FUNCTION_BLOCK FB_WorkerDefGrid_Print_WEU EXTENDS FB_WorkerDefGrid IMPLEMENTS I_PrintSubsystem
VAR_INPUT
  nPrintPos             : DINT;   // Absolute printing position [SubPx]
  fMasterSpeed          : LREAL;  // Speed [m/s]
  bHardwareSync         : BOOL;   // hw sync signal (chenerates a triger internally)
  bHardwareHold         : BOOL;   // hw hold signal
  fPrintStartOffset     : LREAL;  // X-Shift StartOffset from Module reference (configurative PU/PM/PG/PA ADS offset) [m]
  fPrintYOffset         : LREAL;  // Y-Shift
  // fine alignement live parameter
  fPUElevation          : LREAL;  // PU distance from substrate [m]
END_VAR
VAR
  // print
  // - references
  _pAdsPg            : POINTER TO ST_ADS_PG;      // pg ads reference (for pa)
  // - instances
  fbPs               : FB_PS_Grid;
  fbPa               : FB_PA;
  fB_PcAdapter       : FB_PC_Adapter;
  
  // grid specific
  // - references
  _iParamMediator    : I_ParamMediator;
  // - settings
  sDefGridSettings   : ST_DefGridSettings; 
  // - state 
  fCurrentColumnPos  : LREAL; // Currently column position
  fCurrentPreCharge  : LREAL; // Currently to be precharged
  nChargedColumns    : UDINT; // Already charged columns


  // print corrections
  nPointCorrections  : UDINT;     // number of registered point correction handler
  iPointCorrections  : ARRAY[1..nC_NUM_POINTCORRECTIONS] OF I_GridPointCorrection;  // point corrections
  
  // - Time of flight correction of droplets
  fbDropSpeedComp    : FB_DropSpeedComp;
  //
  _pAdsCam           : POINTER TO ST_ADS_CAMERA;  // camera interface PUC
  // - global shifts (applied globally and not on every single point (calcualted based on all CT points))
  _fDxGlobalShift    : LREAL;
  _fDyGlobalShift    : LREAL;

  // settings or helper
  _fPrintStartOffset : LREAL;   // internal print start offset (distance Cam -> PG1 + PG Offset + PU offset)
  _nPosX0            : DINT;    // X0 for last attached CT (detected postion)
  _nPosXS            : DINT;    // XS for last attached CT (shifted print start position)
  _nPosXDelta        : DINT;    // Shift value X0 -> XS
  _fPosY             : LREAL;   // Y shift for last attached CT
  _nPosDeltaToPrint  : DINT;    // delta pos in [SbuPx] from attach to print
  _sCurrentImgDepth  : LREAL;   // Job: current image length [m]
  _bEndless          : BOOL;    // Job: endless
  _bPaStarted        : BOOL;
  _bPaStartRequested : BOOL;
  _sJobDef           : BOOL;
  fBStartTimeout     : TON;
  rTrigHwSync        : R_TRIG;
  _bForceDefGridOff  : BOOL;    // force deformation grid stream to ph off (send 0)
  
  (*grid limit*)
  _fLimitCorrectionX : LREAL;     // correction limit in y (abs) [px]
  _fLimitCorrectionY : LREAL;     // correction limit in y (abs) [px]
    
  (*Messaging*)
  (*we could implement a message handler for ST_ADS_PG message interface*)

END_VAR

VAR PERSISTENT
  _fColumnsToPrecharge : LREAL := nC_COLUMNS_TO_PRECHARGE;
  _fStartShiftOffset   : LREAL := fC_START_SHIFT_OFFSET;
  _fStartShiftFactor   : LREAL := fC_START_SHIFT_FACTOR;
END_VAR

VAR CONSTANT
  iC_NUM_MSG               : UDINT := 5;
  nC_COLUMNS_TO_PRECHARGE  : LREAL := 2.1;
  fC_GRIDPOINT_STREAM_TIME : LREAL := 0.0025;     // time to stream one point [s]
  fC_START_SHIFT_FACTOR    : LREAL := -2.4E-2;
  fC_START_SHIFT_OFFSET    : LREAL := -1.0E-2;
  nC_NUM_POINTCORRECTIONS  : UDINT := 5;
END_VAR

(*
DOC:
What will be different to FB_WorkerDefGrid_Print of DMAX
- Re-Sync StartPosDetect interface with optional camera data (y-shift)
  Clear with Attach(), security clearance
- (maybe not needed) Stream grid faster to PC (we have no break for switching the CT in endless)
- New PDI StartPostion update (+print start only for first CT) --> send to NIOS or hw buffer
- PDI GridPoint stream
- New PDI PrintingLength update (after last streamed point)
- Other rules for Worker position calculation
*)

PROPERTY aPaState : STRING
GET
aPaState := fbPa.aPaState;
END_GET
END_PROPERTY

METHOD PROTECTED  Attach : BOOL
VAR_INPUT
  iCT              : I_CT;                         (*container at triggered event position*)
END_VAR
Attach:=FALSE;

IF SUPER^.Attach(iCT:=iCT) THEN
  // Additional worker checks
    // - job is valid?
  IF _pAttachedCt^.pJob = 0 OR NOT _bJobActive THEN
    Release(iCT:=iCT);
    RETURN;   // do not print
  
  // CT valid & CT present
  ELSIF NOT _pAttachedCt^.bValid OR NOT _pAttachedCt^.bProductPresent THEN
    Release(iCT:=iCT);
    RETURN;   // do not print
  
  // Ignore start due to hardware hold  
  ELSIF bHardwareHold THEN
    _pAttachedCt^.setError(ErrDef:=EC_Print.ecPaAbortHold, Src:=_pEcSrc^);
    Release(iCT:=iCT);
    RETURN;   // do not print
  
  // - OK attach
  ELSE
    Attach := TRUE;
	END_IF
  
  
  //Prepare print station
  sDefGridSettings := _iParamMediator.sDeformationGridSetttings; // or get from CT (but needs to be set even if WorkerDeformation is not enabled) _pAttachedCt^.sDefGridSettings;
  // fix some potential errors
  IF sDefGridSettings.nGridPitchX = 0 THEN sDefGridSettings.nGridPitchX :=1024; LogError(F_concat2('grid not configured, set default nGridPitchX=',TO_STRING(sDefGridSettings.nGridPitchX))); END_IF
  IF sDefGridSettings.nGridPitchY = 0 THEN sDefGridSettings.nGridPitchY :=1024; LogError(F_concat2('grid not configured, set default nGridPitchY=',TO_STRING(sDefGridSettings.nGridPitchY))); END_IF
  
  nChargedColumns := 0;
  fbPs.bPrintEnable := iCT.bValid AND iCT.bProductPresent;
  fbPs.setGrid(sGrid:=sDefGridSettings);
  _fDxGlobalShift := _pAttachedCt^.fDxShift;
  _fDyGlobalShift := _pAttachedCt^.fDyShift;

  //Start print, PA should be in READY or DONE
  
  // Set X print position
  _nPosX0 :=    _pAttachedCt^.getPosX0(nPosDomain:=E_PosDomain.master_pos)
              //- General Shift
              - F_MeterToSubPixel(fbDropSpeedComp.fDropPlacementError, _fPrintResolution*_fSubPxResolution); // - drop compensation*)
  _nPosXDelta := F_MeterToSubPixel(_fPrintStartOffset, _fPrintResolution*_fSubPxResolution); // + PG/PA Shift (additional PG offset 0 for firstLine)
  
  IF GVL_Deformation.bC_UseGlobalGridShift THEN
    _nPosXDelta := _nPosXDelta + FC_LREAL_TO_DINT(_fDxGlobalShift);                  // + global shift from grid points
  END_IF

  _nPosXS := _nPosX0 + _nPosXDelta;
  fB_PcAdapter.setPrintStartPos(nX0:=_nPosXS);
  
  // Set Y print position
  _fPosY := fPrintYOffset;
  IF GVL_Deformation.bC_UseGlobalGridShift THEN
    _fPosY := _fPosY + _fDyGlobalShift;    // + global shift from grid points
  END_IF
  fB_PcAdapter.setPrintYShift(nYShift:=FC_LREAL_TO_DINT(_fPosY));

  // check
  IF _nPosXS < nPrintPos THEN
    LogWarning(Msg:=F_Concat4('Print start position:', TO_STRING(_nPosXS) ,' < Encoder position:', TO_STRING(nPrintPos)));
	END_IF
  
  // save current distance to print position
  _nPosDeltaToPrint := _nPosXS - iCT.GetPos(nPosDomain:=E_PosDomain.master_pos) - _nPosX0;
  checkGridTiming();
  
  
  IF NOT fbPa.bPrinting THEN   // fB_PcAdapter.bAllPrinting
    IF NOT fbPa.printStart() THEN
      LogError(Msg:='PA not ready to start at attach');
      Release(iCT := iCT);
    ELSE
      _bPaStarted := FALSE;
      _bPaStartRequested := TRUE;
      Attach:=TRUE;
    END_IF
  ELSE
    // update start postion if it was already started (endless)
    {warning 'TODO: implement print restart in endless'}
    //fbPa.restartPrint();
    Attach:=TRUE;
  END_IF
  
  // debug log
  LogLvl(Lvl:=E_LogSeverity.Debug, F_Concat4('printStart: at XS:', TO_STRING(_nPosXS), ' ', _pAttachedCt^.print(0)));  // print container
  IF GVL_Deformation.bC_UseGlobalGridShift THEN
    LogLvl(Lvl:=E_LogSeverity.Debug, F_Concat4(
                                        F_Concat3('> XS = X0(', TO_STRING(_pAttachedCt^.GetPosX0(nPosDomain:=E_PosDomain.master_pos)), ')'),
                                        F_Concat3(' + shDx(', TO_STRING(_fDxGlobalShift), ')'),
                                        F_Concat3(' + shStartOffs(', TO_STRING(F_MeterToSubPixel(_fPrintStartOffset,_fPrintResolution*_fSubPxResolution)), ')'),
                                        F_Concat3(' - shDropComp(', TO_STRING(F_MeterToSubPixel(fbDropSpeedComp.fDropPlacementError,_fPrintResolution*_fSubPxResolution)), ')')
                                     ));
  ELSE
    LogLvl(Lvl:=E_LogSeverity.Debug, F_Concat3(
                                        F_Concat3('> XS = X0(', TO_STRING(_pAttachedCt^.GetPosX0(nPosDomain:=E_PosDomain.master_pos)), ')'),
                                        F_Concat3(' + shStartOffs:', TO_STRING(F_MeterToSubPixel(_fPrintStartOffset,_fPrintResolution*_fSubPxResolution)), ')'),
                                        F_Concat3( ' - shDropComp:', TO_STRING(F_MeterToSubPixel(fbDropSpeedComp.fDropPlacementError,_fPrintResolution*_fSubPxResolution)), ')')
                                     ));
  END_IF
  
  
ELSE
  // parent attach failed case
END_IF
END_METHOD

PROPERTY bPausePrintCanEx : BOOL
GET
bPausePrintCanEx := FALSE; //Not implemented
END_GET
END_PROPERTY

PROPERTY bPcEnabled : BOOL
GET
bPcEnabled := fB_PcAdapter.bPcEnable;
END_GET
END_PROPERTY

PROPERTY bPrintEnabled : BOOL
GET
bPrintEnabled := _bEnable;
END_GET
END_PROPERTY

PROPERTY bPrintError : BOOL
GET
bPrintError := bError; // Worker error 
                  // or fB_PcAdapter.bError
END_GET
END_PROPERTY

PROPERTY bPrinting : BOOL
GET
bPrinting := fbPa.bPrinting;
END_GET
END_PROPERTY

PROPERTY bPrintReady : BOOL
GET
bPrintReady := fbPa.bReady;
END_GET
END_PROPERTY

PROPERTY bStartPrintCanEx : BOOL
GET
bStartPrintCanEx := fbPa.bStartCanEx;
END_GET
END_PROPERTY

PROPERTY bStopPrintCanEx : BOOL
GET
bStopPrintCanEx := fbPa.bStopCanEx;
END_GET
END_PROPERTY

{attribute 'monitoring':='call'}
PROPERTY bWorkerEnable : BOOL
GET
bWorkerEnable := SUPER^.bWorkerEnable;
END_GET
SET
IF _pAdsPg = 0 THEN
  SUPER^.bWorkerEnable := bWorkerEnable;
ELSE
  // mask worker enable with group enable
  SUPER^.bWorkerEnable := bWorkerEnable AND _pAdsPg^.bI_Enable;  
END_IF
END_SET
END_PROPERTY

METHOD PRIVATE checkGridTiming : BOOL
VAR
END_VAR
// check for timing problems
IF fMasterSpeed <> 0 THEN

  // - check pre-charge at beginning
  IF _fColumnsToPrecharge * fC_GRIDPOINT_STREAM_TIME * GVL_Deformation.nC_GridRoiRows >= F_SubPixelToMeter(lPosSubPx:=_nPosDeltaToPrint, fResSubPx:=_fPrintResolution*_fSubPxResolution) / fMasterSpeed  THEN
       LogError('Machine too fast for grid stream (for pre-charge at attach)');
  END_IF
  
 // - check charge time needed per columns vs machine speed and grid-sizeY
 IF GVL_Deformation.nC_GridRoiRows * fC_GRIDPOINT_STREAM_TIME >= F_SubPixelToMeter(lPosSubPx:=TO_DINT(sDefGridSettings.nGridPitchX), fResSubPx:=_fPrintResolution) / fMasterSpeed THEN
   LogError('Machine too fast for grid stream (time rows per column)');
 END_IF

END_IF
END_METHOD

(*
  Limit correction to boundaries
  :return: TRUE if limited
*)
METHOD PRIVATE correctionLimit : BOOL
VAR_INPUT
  pPoint : POINTER TO ST_DeformationPointAccurate;
END_VAR
VAR
  bLimited : BOOL;
  nExeedX, nExeedY : LREAL;
END_VAR
// limit point correction to boundaries and inform
IF    pPoint^.dx >= _fLimitCorrectionX    THEN nExeedX := pPoint^.dx; pPoint^.dx := _fLimitCorrectionX;    bLimited:=TRUE; 
ELSIF pPoint^.dx <= -1*_fLimitCorrectionX THEN nExeedX := pPoint^.dx; pPoint^.dx := -1*_fLimitCorrectionX; bLimited:=TRUE;
ELSIF pPoint^.dy >= _fLimitCorrectionY    THEN nExeedY := pPoint^.dy; pPoint^.dy := _fLimitCorrectionY;    bLimited:=TRUE;
ELSIF pPoint^.dy <= -1*_fLimitCorrectionY THEN nExeedY := pPoint^.dy; pPoint^.dy := -1*_fLimitCorrectionY; bLimited:=TRUE;
END_IF
IF bLimited THEN 
  LogLvl(Lvl:=E_LogSeverity.Warning, Msg:=F_Concat5( 'Point=',TO_STRING(pPoint^.index),
                                                     F_Concat5(' c/r(',TO_STRING(pPoint^.col),'/',TO_STRING(pPoint^.row), ') '),
                                                     F_Concat4('dx:', TO_STRING(nExeedX), ' dy:', TO_STRING(nExeedY)),
                                                     ' correction exceeded limit')); 
END_IF
correctionLimit := bLimited;
END_METHOD

METHOD PRIVATE correctionUpdate : BOOL
VAR_INPUT
  pPoint : POINTER TO ST_DeformationPointAccurate;
END_VAR
VAR
  i : UDINT;
END_VAR

// here apply all PU specific corrections
// - mechanical stretch based on temperature extension (if not done in Camera)
// - banana correction
// - Y-shifts of PU
// - trapzedoial correction
// - ...

// global dx/dy correction
//   remove global shift from GridPoints (shifted by PU)
IF GVL_Deformation.bC_UseGlobalGridShift THEN
  pPoint^.dx := pPoint^.dx - _fDxGlobalShift;
  pPoint^.dy := pPoint^.dy - _fDyGlobalShift;
END_IF

// PU Deformation correction
IF GVL_Deformation.bC_UsePUDeformation THEN
  FOR i:=1 TO nPointCorrections DO
    iPointCorrections[i].updateCorrection(pPoint:=pPoint);
  END_FOR
END_IF
END_METHOD

(*
  Max. supported speed [m/s], 0 if not available
*)
{attribute 'monitoring':='call'}
PROPERTY fMaxSpeed : LREAL
GET
VAR
  nSpeedMpMin : DINT;
END_VAR
nSpeedMpMin := SEL(bWorkerEnable AND _pAdsPg <> 0, 0, _pAdsPg^.sI_MaxPrintSpeed.lI_Val);
fMaxSpeed := TO_LREAL(nSpeedMpMin)/60;
END_GET
END_PROPERTY

{attribute 'monitoring':='call'}
PROPERTY fStartShiftFactor : LREAL
GET
fStartShiftFactor := _fStartShiftFactor;
END_GET
SET
_fStartShiftFactor := fStartShiftFactor;
END_SET
END_PROPERTY

{attribute 'monitoring':='call'}
PROPERTY fStartShiftOffset : LREAL
GET
fStartShiftOffset := _fStartShiftOffset;
END_GET
SET
_fStartShiftOffset := fStartShiftOffset;
END_SET
END_PROPERTY

METHOD PROTECTED gridUpdate : BOOL
VAR_INPUT
  bEnableDeformation : BOOL;      // enable correction update, else correction (0/0) is written
END_VAR
VAR
  sPoint : ST_DeformationPointAccurate;
  nRow : UDINT;
  nAvailPoints : UDINT;
  nConvErr : UDINT;
END_VAR
VAR_INST
  nAvailPoints_mem : UDINT;
END_VAR
//TODO: rewrite this method to look cleaner (less if else)
IF sDefGridSettings.nGridSizeX = 0 THEN RETURN; END_IF          // avoid endless loops
IF sDefGridSettings.nGridSizeY = 0 THEN RETURN; END_IF

gridUpdate:=TRUE;

// calculate grid column position
IF sDefGridSettings.nGridPitchX <> 0 THEN
  fCurrentColumnPos := fCtPosition / (sDefGridSettings.nGridPitchX * _fSubPxResolution);   // calc grid column position relative to worker
END_IF

//Check for next correction update 
IF fCurrentColumnPos + _fColumnsToPrecharge > nChargedColumns AND nChargedColumns <= sDefGridSettings.nGridSizeX THEN
  fCurrentPreCharge := fCurrentColumnPos + _fColumnsToPrecharge;
  IF bEnableDeformation THEN 
    // sync deformation points
    WHILE FLOOR(fCurrentPreCharge) > nChargedColumns AND nChargedColumns <= sDefGridSettings.nGridSizeX DO
      nAvailPoints := _pAttachedCt^.nAvailableGridPoints;
      IF nAvailPoints >= sDefGridSettings.nGridSizeY * (nChargedColumns+1) THEN // Complete column available?
        nAvailPoints_mem := 0;
        LogLvl(Lvl:=E_LogSeverity.Debug, Msg:=F_Concat2('Charge CG col: ',TO_STRING(nChargedColumns)));
        FOR nRow := 0 TO sDefGridSettings.nGridSizeY - 1 DO
          // get points
          IF _pAttachedCt^.getDeformationPoint(nCol:=nChargedColumns, nRow:=nRow, sPoint => sPoint) THEN
            // transfer the displacement into a correction
            sPoint.dx := sPoint.dx;   // nothing to change
            sPoint.dy := sPoint.dy;
            
            // apply PU corrections
            correctionUpdate(pPoint:=ADR(sPoint));
            
            // correction limitation
            correctionLimit(pPoint:=ADR(sPoint));
            
            // send point
            IF NOT fbPs.newGridPoint(sPoint:=sPoint) THEN
               LogError(Msg:='stream new point failed');
               gridUpdate:=FALSE;
               RETURN;
            END_IF
          ELSE
            LogError(Msg:='get new grid point failed');
            gridUpdate:=FALSE;
          END_IF
        END_FOR
        
        nChargedColumns := nChargedColumns + 1;
      ELSE
        IF nAvailPoints > nAvailPoints_mem THEN // log once or after every update of new available poinst
          LogError(Msg:='point column expected but not available');
        END_IF
        nAvailPoints_mem := nAvailPoints;
        gridUpdate:=FALSE;
        RETURN;
      END_IF 
    END_WHILE
  ELSE
    // send points with no deformation
    FOR nRow := 0 TO sDefGridSettings.nGridSizeY - 1 DO
        MEMSET(destAddr:=ADR(sPoint), fillByte:=0, n:=SIZEOF(sPoint));
        sPoint.col := TO_DINT(nChargedColumns);
        sPoint.row := TO_DINT(nRow);
        IF NOT fbPs.newGridPoint(sPoint:=sPoint) THEN
           LogError(Msg:='stream new point failed');
           gridUpdate:=FALSE;
           RETURN;
        END_IF
    END_FOR
    nChargedColumns := nChargedColumns + 1;
  END_IF
END_IF
END_METHOD

METHOD InitWorkerPrint : BOOL
VAR_INPUT
  pAdsPg                : POINTER TO ST_ADS_PG;       // pg ads reference (worker prints ads)
  iDefGridParamMediator : I_ParamMediator;            // for deformation settings
  fLimitCorrectionX     : LREAL;                      // correction limit in y (abs) [px]
  fLimitCorrectionY     : LREAL;                      // correction limit in y (abs) [px]
END_VAR
IF NOT bInitialized            THEN LogError('Base Worker not initialized! call init() before'); RETURN; END_IF
IF pAdspg = 0 THEN LogError('InitWorkerPrint: invalid parameter proviced'); RETURN; END_IF
IF iDefGridParamMediator = 0   THEN bInitialized := FALSE; LogError('Invalid parameter, no valid param mediator'); RETURN; END_IF

// Worker specific init
_pAdsPg := pAdsPg;
_iParamMediator := iDefGridParamMediator;

_fLimitCorrectionX := ABS(fLimitCorrectionX);
_fLimitCorrectionY := ABS(fLimitCorrectionY);

// Print Aggregate
fbPa.bSyncAfterDone := FALSE;
fbPa.init(iPcAdapter := fB_PcAdapter, iPsInterface := fbPs);
END_METHOD

METHOD mJobPause
END_METHOD

METHOD   mJobStart
VAR_INPUT
	sJobDef	: CalmarCompPrint.I_JobDefinition;
END_VAR
// Config workers static variables
_fCtSecurityReleasePos := F_MeterToSubPixel(fPosMeter:=sJobDef.fImageDepth/1000 + fC_MIN_SHEET_GAP, fResoSubPx:=_fPrintResolution*_fSubPxResolution);

IF NOT bWorkerEnable THEN RETURN; END_IF  // only if enabled

fbPa.jobStart();

_sCurrentImgDepth := sJobDef.fImageDepth/1000;
_bEndless := sJobDef.isEndless();

_bJobActive := TRUE;
END_METHOD

METHOD  mJobStop
VAR_INPUT
	sStatus	: CalmarCompPrint.I_JobStatus;
END_VAR
fbPa.jobStop();
_bJobActive := FALSE;
_bPaStarted := FALSE;
_bPaStartRequested := FALSE;
END_METHOD

METHOD mProduced
VAR_INPUT
	(* current progress*)
	sProgress	: CalmarCompPrint.I_JobProgress;
END_VAR
END_METHOD

METHOD RegisterGridCorrection : BOOL
VAR_INPUT
  iGridCorrection : I_GridPointCorrection;
END_VAR
VAR
  i : UDINT;
END_VAR
IF iGridCorrection = 0 THEN LogError('registerGridCorrection: ivalid interface, ignore'); RETURN; END_IF
IF nPointCorrections >= nC_NUM_POINTCORRECTIONS THEN LogError('registerGridCorrection: too many corrections registred, ignore'); RETURN; END_IF

nPointCorrections := nPointCorrections + 1;
iPointCorrections[nPointCorrections] := iGridCorrection;
END_METHOD

METHOD registerPc : BOOL
VAR_INPUT
  iNewPC : I_PC;
END_VAR
registerPc := fB_PcAdapter.registerPc(iNewPC := iNewPC);
END_METHOD

METHOD registerPh : BOOL
VAR_INPUT
    iPH : I_PH;
    iNewCG : I_Correction_Grid;   // correction grid interface
END_VAR
//Attach head to print station
IF iPH <> 0 THEN
  fbPs.registerCG(iNewPh:=iPH, iNewCG:=iNewCG);
END_IF
END_METHOD

METHOD PRIVATE sim
END_METHOD

METHOD PRIVATE updateWorkerPosition
VAR_INPUT
END_VAR
// Update only without attached container
IF _pAttachedCt = 0 THEN RETURN; END_IF

//Start offset update
IF _fPrintStartOffset <> (fPrintStartOffset + _iWorkerParams.fDetectToRefPos) THEN //Worker position changed
  _fPrintStartOffset := fPrintStartOffset + _iWorkerParams.fDetectToRefPos;
END_IF

//Worker position update
IF _fWorkerPosition <> (_fPrintStartOffset + (_fStartShiftOffset + _fStartShiftFactor * fMasterSpeed)) THEN   // Worker position changed (camera settings change)
  // WorkerPosition = PrintStart offset - pre-start offset
  fPosition := _fPrintStartOffset + (_fStartShiftOffset + _fStartShiftFactor * fMasterSpeed);
END_IF
END_METHOD

METHOD  work
VAR
  bDeformErr : BOOL;
  nDeformStep : E_DeformationStep;
END_VAR
IF _iWorkerParams = 0 OR _iParamMediator = 0 THEN F_Report_Error(ErrType:=EN_REPORT_ERROR_TYPE.Report_Error_0Pointer); RETURN; END_IF
bError := FALSE; nError := 0;

updateWorkerPosition();  // calculate and set worker position

SUPER^.work();

(*Print correction*)
fbDropSpeedComp(fMasterSpeed:=fMasterSpeed, fDropTravelDistance:=fPUElevation);


(*Update virtual encoder on all controller boards*)
fB_PcAdapter.setEncoderPos(nPrintPos);
fB_PcAdapter();

(*Call print aggregate*)
rTrigHwSync(CLK:=bHardwareSync); 
IF rTrigHwSync.Q THEN fbPa.sync(); END_IF   // external sync cmd
fbPa.bHold := bHardwareHold;                // external hw hold, NOTE: this stop the current print iPC.stop()
fbPa();

fBStartTimeout(IN:=_bPaStartRequested, PT := T#60MS);

IF _pAttachedCt <> 0 AND bWorkerEnable THEN // Work only with attached container
  
  // check for generic error
  IF _pAttachedCt^.bValid AND bHardwareHold THEN
    // abort during printing
    _pAttachedCt^.setError(ErrDef:=EC_Print.ecPaAbortHold, Src:=_pEcSrc^);
  END_IF

  // Grid update
  bDeformErr := _pAttachedCt^.getDeformationStatus(eDStep=>nDeformStep);
  IF NOT bDeformErr AND nDeformStep >= E_DeformationStep.gridStarted AND NOT _bForceDefGridOff THEN 
    IF NOT gridUpdate(bEnableDeformation:=TRUE) THEN
      _pAttachedCt^.AbortDeformation(sReason:='deformation point update failed', Src:=_pEcSrc^);
      //Release(iCT:=_pAttachedCt^);
    END_IF
  ELSE
    // not started or error already --> erase deformation points and send no correction points
    IF NOT gridUpdate(bEnableDeformation:=FALSE) THEN
      _pAttachedCt^.AbortDeformation(sReason:='deformation point update failed', Src:=_pEcSrc^);
      //Release(iCT:=_pAttachedCt^);
    END_IF
  END_IF

  // PA control
  IF _bPaStartRequested THEN
    IF fbPa.bPrinting THEN
      _bPaStarted := TRUE;
      _bPaStartRequested := FALSE;
    ELSIF fBStartTimeout.Q THEN //Stop print at timeout to make ready for next container
      _bPaStarted := FALSE;
      _bPaStartRequested := FALSE;
      fbPa.printStop();
      _pAttachedCt^.setError(ErrDef:=EC_Print.ecPaStartErr, Src:=_pEcSrc^);
      Release(_pAttachedCt^);
		END_IF
  ELSIF _bPaStarted THEN
    //Release container when all points have been processed
    IF fbPa.bDone OR fbPa.bStop THEN
      _bPaStarted := FALSE;
      Release(_pAttachedCt^);
    (*ELSIF fbpa.bError THEN
      _pAttachedCt^.setError(ErrDef:=EC_Print.ecPaPrintErr, Ident:=0);
      Release(_pAttachedCt^);*)
    ELSE
      // still printing (endless or not yet done)
      IF _bEndless AND nChargedColumns >= sDefGridSettings.nGridSizeX THEN
        // in endless release if grid was streamed
        {warning 'TODO: send real PrintLength _pAttachedCt^.bPrintLength'} 
        Release(_pAttachedCt^);
			END_IF
    END_IF 
	END_IF
END_IF  


// forward pa state to pg ads
IF _pAdsPg <> 0 THEN
  _pAdsPg^.aO_State := fbPa.aPaState;
  _pAdsPg^.lO_Error := nError; 
  _pAdsPg^.bO_Error := bError;
END_IF

// logging config
fbPa.LogLevel := LogLevel;
fB_PcAdapter.LogLevel := LogLevel;

sim();
END_METHOD

END_FUNCTION_BLOCK

(* stored: Version 1.1.0.1, ProductVersion 3.1.4024.11
   POU FB_WorkerDefGrid_Print_WEU: Id {a51f391c-3039-4bd9-921c-4da39276f1e6}, SpecialFunc None
   Folder I_PrintStatusClient: Id {e7b8ed8a-f644-4467-ad9b-c45a3bfc8aa7}
   Folder I_PrintSubsystem: Id {6caba1d4-15ea-4dff-b84f-85eedc71ff04}
   Property aPaState: Id {8cd6fce7-6a00-4fb3-a4a5-292eaf4f7f86}
   Get Get: Id {770c0a62-8e79-4bff-acf2-d69ceee7eea5}
   Method Attach: Id {04289869-54be-4698-97f6-46fa0259e7dd}
   Property bPausePrintCanEx: Id {90a0cfcd-d04f-44f8-8556-390310f6346d}
   Get Get: Id {c2aceddc-dd50-49ed-8b3e-551468a705b8}
   Property bPcEnabled: Id {7e86c0b9-f8cf-4434-9add-45495a769294}
   Get Get: Id {71f8a8db-9bcc-441f-a75b-c719625a0bf4}
   Property bPrintEnabled: Id {08effb3f-d924-408a-941d-ff2b13a9a83e}
   Get Get: Id {0711cb07-c232-47ba-a2f6-9293867dfecf}
   Property bPrintError: Id {7093e9ca-6584-42d4-86f4-897ee7f3c2d8}
   Get Get: Id {92d6f28b-8c51-4dde-b836-d1c779011e1f}
   Property bPrinting: Id {ada463a7-669b-43d2-b48c-8fd4f72b7fbc}
   Get Get: Id {17171856-ee80-4eb4-bc57-ce5faab30d99}
   Property bPrintReady: Id {4e6bc301-4620-4318-89c9-ab4150116aea}
   Get Get: Id {7704a91a-fa13-46ae-ab5b-e4d9875d106b}
   Property bStartPrintCanEx: Id {113bf46a-17a0-4262-aeb3-2210e7d207b3}
   Get Get: Id {b1e937bf-f460-408f-88da-2672d9b61adc}
   Property bStopPrintCanEx: Id {a62f9288-4559-4001-90c5-02b46605889a}
   Get Get: Id {16ab9ebf-f44a-40a5-bbfb-aaf539ba6362}
   Property bWorkerEnable: Id {671684a2-d248-4dc0-bd0b-0fe74a1f3006}
   Get Get: Id {091237bc-ae12-4dc9-a493-c0a6c2dac5b7}
   Set Set: Id {3d6b8fca-3946-4af7-b7c7-9f16646edacf}
   Method checkGridTiming: Id {82d69843-5ea3-4291-ac3c-a02d205e898c}
   Method correctionLimit: Id {9e9550be-5844-456c-8fe6-7fcc69bb324c}
   Method correctionUpdate: Id {14cecb46-16e0-4f17-918f-ce5692924079}
   Property fMaxSpeed: Id {e93ac3c2-7afb-43cc-a5a4-ff642c3d646c}
   Get Get: Id {950b9b28-2b18-46b2-acf5-2db9b914a945}
   Property fStartShiftFactor: Id {76fc8cfe-283f-4ec4-a887-b19a187f997f}
   Get Get: Id {190c48b1-4bf5-49c7-9e8c-05ddb0715765}
   Set Set: Id {cf520747-e9c6-4c48-9245-8466cce47ffc}
   Property fStartShiftOffset: Id {b4313e10-b46d-4236-a465-4c511fe68aa8}
   Get Get: Id {c259f77b-dbd1-44c9-aad3-424b6b4371d0}
   Set Set: Id {9edee42a-9a9a-460f-9332-fa95a49308cd}
   Method gridUpdate: Id {bdd499b9-f393-484d-a6e4-c9de3446cbae}
   Method InitWorkerPrint: Id {725b4782-e9a9-4287-9bbe-5c631e47969c}
   Method mJobPause: Id {94f00e92-8a20-43a9-9616-e560f3ba3770}
   Method mJobStart: Id {89edfdce-4466-46a7-a112-cf11e587d110}
   Method mJobStop: Id {05477037-33e9-4fec-9299-59aab145ce38}
   Method mProduced: Id {09c64151-c707-4a94-bc62-7cee61472f96}
   Method RegisterGridCorrection: Id {d479508c-6130-4d9d-9335-d417617a9a10}
   Method registerPc: Id {4776f3c2-c3e1-4f90-b8f6-3a06b4691e15}
   Method registerPh: Id {6c4c9059-69e5-4f42-ba66-a286f447450f}
   Method sim: Id {60553fe4-14ee-48fc-82de-1d9573b5e2ec}
   Method updateWorkerPosition: Id {5207464a-bb68-4cfe-bdd9-989eb1679161}
   Method work: Id {67970e4d-2ad9-4f9e-8bde-95cb4f3188e8} *)
